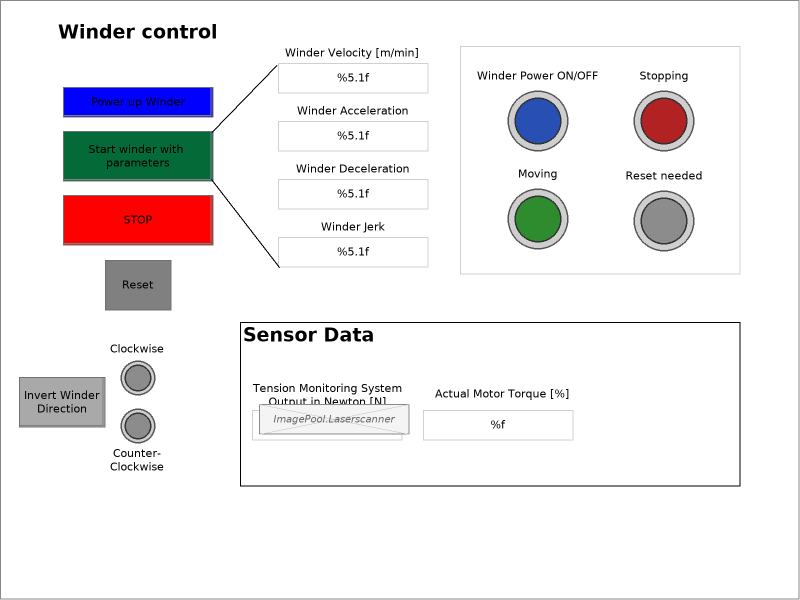
VISUALIZATION Winder_control  // 800x600
    Textfield (460,46 280x228)
    Textfield (240,322 500x164), "Sensor Data"
    Label (52,17 172x30), "Winder control"
    Textfield (278,63 150x30), "%5.1f", text variable: GVL_Axis.rWinderVelocity
        OnMouseClick: write the text variable via VisuDialogs.Numpad, min 2.7, max 15
    Label (277,38 150x30), "Winder Velocity [m/min]"
    Textfield (278,121 150x30), "%5.1f", text variable: GVL_Axis.rWinderAcceleration
        OnMouseClick: write the text variable via Default
    Label (278,96 150x30), "Winder Acceleration"
    Textfield (278,237 150x30), "%5.1f", text variable: GVL_Axis.rWinderJerk
        OnMouseClick: write the text variable via Default
    Textfield (278,179 150x30), "%5.1f", text variable: GVL_Axis.rWinderDeceleration
        OnMouseClick: write the text variable via Default
    Label (278,154 150x30), "Winder Deceleration"
    Label (278,212 150x30), "Winder Jerk"
    Button (63,87 150x30), "Power up Winder", colour toggle: GVL_HMI.bButtonWinderPower
        toggle GVL_HMI.bButtonWinderPower
    Button (63,131 150x50), "Start winder with parameters", colour toggle: GVL_HMI.bButtonStartWinder
        OnMouseDown: execute { GVL_HMI.bButtonStartWinder := TRUE; }
        OnMouseUp: execute { GVL_HMI.bButtonStartWinder := FALSE; }
    Button (63,195 150x50), "STOP", colour toggle: GVL_HMI.bButtonStopWinder
        OnMouseDown: execute { GVL_HMI.bButtonStopWinder := TRUE; }
        OnMouseUp: execute { GVL_HMI.bButtonStopWinder := FALSE; }
    Button (105,260 66x50), "Reset", colour toggle: GVL_HMI.bButtonResetWinder
        OnMouseDown: execute { GVL_HMI.bButtonResetWinder := TRUE; }
        OnMouseUp: execute { GVL_HMI.bButtonResetWinder := FALSE; }
    Line (212,132) (277,65)
    Line (211,179) (279,267)
    Lamp1 (503,86 70x70), variable: GVL_Axis.bStatusPower, style: Lamp-Lamp1-Blue
    Label (463,61 150x30), "Winder Power ON/OFF"
    Lamp1 (503,184 70x70), variable: GVL_Axis.bStateCM, style: Lamp-Lamp1-Green
    Label (463,159 150x30), "Moving"
    Group (589,61 150x195)
        Lamp1 (40,25 70x70), variable: GVL_Axis.bStateStopping, style: Lamp-Lamp1-Red
        Label (0,0 150x30), "Stopping"
        Lamp1 (40,125 70x70), variable: GVL_Axis.bStateErrorStop, style: Lamp-Lamp1-Gray
        Label (0,100 150x30), "Reset needed"
    Textfield (252,410 150x30), "%i", text variable: GVL.iTensionMonitoringData
    Label (246,380 163x30), "Tension Monitoring System Output in Newton [N]"
    Button (19,377 86x50), "Invert Winder Direction", colour toggle: GVL_HMI.bButtonWinderDirection
        toggle GVL_HMI.bButtonWinderDirection
    Lamp1 (118,358 40x40), variable: GVL_HMI.bButtonWinderDirection, style: Lamp-Lamp1-Gray
    Lamp1 (118,406 40x40), variable: GVL_HMI.bButtonNotWinderDirection, style: Lamp-Lamp1-Gray
    Label (95,334 84x30), "Clockwise"
    Label (95,445 84x30), "Counter- Clockwise"
    Textfield (237,275 231x45), "!!New Motion Parameter detected!! Click 'Start winder' to update Parameters", colour toggle: GVL_Axis.bNewMotionParameter
    Textfield (423,410 150x30), "%f", text variable: GVL_HMI.ActTorque
    Label (421,379 163x30), "Actual Motor Torque [%]"
    Image (259,404 150x30), image: ImagePool.Laserscanner
END_VISUALIZATION

(* stored: Version 1.1.0.1
   Visu Winder_control: Id {64a93884-b594-4d4d-81c2-aab08f44ffa1} *)
